//-----------------------------------------------------------------------------------------------------
//																
//									 	Tkmatik sp z o.o.
//
//	Name					:		FB_Save
//	Author					:		AM
//	Release Date			:		12.01.2022
//	Current ver				:		v 0.1
// 	Last correction 		:		12.01.2022
// 
//	Description				:
//		Special FB for saving structures to CSV files						
//
//	Requared hardware		:
//
// 	Configuration			:
//
//
//-----------------------------------------------------------------------------------------------------

FUNCTION_BLOCK FB_RecipeSaveCSV

VAR_INPUT
	bExecute							: BOOL := FALSE;(* Rising edge starts program execution *)
	sFilePath							: T_MaxString;(* CSV destination file path and name *)
//	database							: POINTER TO STRING(255);	
	nRows          						: UDINT;                // Liczba wierszy
    nCols          						: UDINT; 
	database							: POINTER TO STRING(255);//ARRAY[0..MAX_PARAMS_VARIABLES_COUNT-1] OF STRING(255);
END_VAR
VAR CONSTANT
	MAX_CSV_FIELD_LENGTH				: UDINT	:= 255;	
END_VAR
VAR_IN_OUT
END_VAR

VAR
	
	sNetId			: T_AmsNetId := '';	(* TwinCAT system network address *)
	sCSVLine		: T_MaxString := '';(* Single CSV text line (row, record), we are using string as record buffer (your are able to see created fields) *)
	sCSVField		: T_MaxString := '';(* Single CSV field value (column, record field) *)
	nRow	 		: UDINT 	:= 0;(* Row number (record) *)
	nColumn			: UDINT 	:= 0;(* Column number (record field) *)
	hFile			: UINT		:= 0;(* File handle of the source file *)
	step			: DWORD 	:= 0;
	fbFileOpen		: FB_FileOpen;(* Opens file *)
	fbFileClose		: FB_FileClose;(* Closes file *)
	fbFilePuts		: FB_FilePuts;(* Writes one record (line) *)
	fbWriter		: FB_CSVMemBufferWriter;(* Helper function block used to create CSV data bytes (single record line) *)
	rtExecute		:	R_TRIG;                         //	Rtrig for start



END_VAR
VAR_OUTPUT                                                                                  
	bBusy												:	BOOL;                           //	FB is Busy
	bDone												:	BOOL;                           //	Load cycle done, DATA actual 
	bError												:	BOOL;                           //	Flag error
	nErrId												:	UDINT;                          //	Error ID
END_VAR

rtExecute(CLK:=bExecute);
IF (NOT bExecute) THEN
	bDone												:=	FALSE;
END_IF

CASE step OF
	0:	(* Wait for rising edge at bWrite variable *)
		IF rtExecute.Q THEN
			bBusy 	:= TRUE;
			bError	:= FALSE;
			nErrId	:= 0;
			hFile	:= 0;
			nRow	:= 0;
			nColumn	:= 0;
			step 	:= 1;
		END_IF

	1:	(* Open source file *)
		fbFileOpen(  bExecute := FALSE  );
		fbFileOpen( sNetId := sNetId, sPathName := sFilePath, nMode := FOPEN_MODEWRITE OR FOPEN_MODETEXT,(* Open file in TEXT mode! *)
					ePath := PATH_GENERIC, bExecute := TRUE );
		step := 2;

	2:(* Wait until open not busy *)
		fbFileOpen( bExecute := FALSE, bError => bError, nErrID => nErrID, hFile => hFile );
		IF NOT fbFileOpen.bBusy THEN
			IF NOT fbFileOpen.bError THEN
				step := 3;
			ELSE(* Error: file not found? *)
				step := 100;
			END_IF
		END_IF

	3:(* Convert one PLC record to CSV format *)
		sCSVLine := '';
		fbWriter.eCmd := eEnumCmd_First;(* Write first field value *)
		IF nRow <= nRows THEN

			FOR nColumn := 0 TO nCols BY 1 DO
 
				sCSVField := STRING_TO_CSVFIELD( database[ nRow ], FALSE );(* TODO: Get field value from your application *)

				(* Add new field to the record buffer *)
				fbWriter( 	pBuffer := ADR( sCSVLine ), cbBuffer := SIZEOF( sCSVLine ) - 1, putValue := sCSVField, pValue := 0, cbValue := 0,
							bCRLF := ( nColumn = nCols ) );(* bCRLF == TRUE => Write CRLF after the last field value *)
				IF fbWriter.bOk THEN
					fbWriter.eCmd := eEnumCmd_Next;(* Write next field value *)
				ELSE(* Error *)
					step := 100;
					RETURN;
				END_IF

			END_FOR(* FOR nColumn := 0... *)

			(* FB_FilePuts adds allready CR (carriage return) to the written line.
			We have to replace the $R$L characters with $L character to avoid double CR. *)
			IF RIGHT( sCSVLine, 2 ) = '$R$L' THEN
				sCSVLine := REPLACE( sCSVLine, '$L', 2, LEN( sCSVLine ) - 1 );
			END_IF

			nRow := nRow + 1;(* Increment number of created records (rows) *)
			step := 4;(* Write record to the file *)

		ELSE(* All rows written => Close file *)
			step := 10;
		END_IF

	4:	(* Write single text line *)
		fbFilePuts( bExecute := FALSE );
		fbFilePuts( sNetId := sNetId, hFile := hFile, sLine := sCSVLine, bExecute := TRUE );
		step := 5;

	5:(* Wait until write not busy *)
		fbFilePuts( bExecute := FALSE, bError => bError, nErrID => nErrID );
		IF NOT fbFilePuts.bBusy THEN
			IF NOT fbFilePuts.bError THEN
				step := 3;(* Write next record *)
			ELSE(* Error *)
				step := 100;
			END_IF
		END_IF

	10:	(* Close source file *)
		fbFileClose( bExecute := FALSE );
		fbFileClose( sNetId := sNetId, hFile := hFile, bExecute := TRUE );
		step := 11;

	11:(* Wait until close not busy *)
		fbFileClose( bExecute := FALSE, bError => bError, nErrID => nErrID );
		IF ( NOT fbFileClose.bBusy ) THEN
			bDone	:= TRUE;
			hFile := 0;
			step := 100;
		END_IF

	100: (* Error or ready step => cleanup *)
		IF ( hFile <> 0 ) THEN
			step := 10; (* Close the source file *)
		ELSE
			bBusy := FALSE;
			step := 0;	(* Ready *)
		END_IF

END_CASE

END_FUNCTION_BLOCK

(* stored: Version 1.1.0.1, ProductVersion 3.1.4026.13, FileIdentifier ff74270a61b01ff97e890e3b3b49666747c0ff50, FileSignature 123bd5bc833d51b1ee5e3c4dc5e434ecd6c7b7655c7a7edac67670c896dadd262df57dd35ede32a8e7a26af63bc759830ee6538a8ee828066dbfd7e4952b42c6348e3030973c3838e61a6c914bc0d95ac4b58ef5f27d18ac4b034d8cc22d26d7df223b03632b5c0ca14ae3b356567ca099f8779033456f4506a237f82bdd7b1a0bb5d2b2d48d3b4a40436ab71425ee77187aa62105ca4c326d38a78db0cfac18cdd635f6ed35b152f65787ccb769f3741f35d65b4b215f723b3f58421bac58134b1830d827bde1a5518ed8e42affb9d8f940f33b47b4e4e6e9d0aa799b587b03de5ea51e1bc8a2810330394cb7c44ca4653bf358b100e58c2b4f49113d4ed01f
   POU FB_RecipeSaveCSV: Id {b281a86b-4121-439e-8d81-60c40caede61}, SpecialFunc None *)
